FUNCTION_BLOCK FB_StationPLC IMPLEMENTS I_Device, I_Test
VAR_INPUT
END_VAR
VAR_OUTPUT
END_VAR
VAR
END_VAR


// Used to Handhsake Test Controller IPC and Station PLC
mTestStart();
mTestStop();

{warning 'add method implementation '}
METHOD mDeviceComm : BOOL
END_METHOD

{warning 'add method implementation '}
METHOD mDeviceEnable : BOOL
END_METHOD

{warning 'add method implementation '}
METHOD mDeviceHeartbeat : BOOL
END_METHOD

{warning 'add method implementation '}
METHOD mDeviceReset : BOOL
END_METHOD

{warning 'add method implementation '}
METHOD mDeviceStatus : E_DeviceStatus
END_METHOD

{warning 'add method implementation '}
METHOD mTestComp : BOOL
END_METHOD

{warning 'add method implementation '}
METHOD mTestFault : BOOL
END_METHOD

{warning 'add method implementation '}
METHOD mTestResult : BOOL
END_METHOD

{warning 'add method implementation '}
METHOD mTestStart : BOOL
END_METHOD

{warning 'add method implementation '}
METHOD mTestStop : BOOL
END_METHOD

{warning 'add property implementation'}
PROPERTY pDeviceCommOK : BOOL
GET
END_GET
SET
END_SET
END_PROPERTY

{warning 'add property implementation'}
PROPERTY pDeviceEnableCmd : BOOL
GET
END_GET
SET
END_SET
END_PROPERTY

{warning 'add property implementation'}
PROPERTY pDeviceEnabled : BOOL
GET
END_GET
SET
END_SET
END_PROPERTY

{warning 'add property implementation'}
PROPERTY pDeviceFaulted : BOOL
GET
END_GET
SET
END_SET
END_PROPERTY

{warning 'add property implementation'}
PROPERTY pDeviceReady : BOOL
GET
END_GET
SET
END_SET
END_PROPERTY

{warning 'add property implementation'}
PROPERTY pDeviceReset : BOOL
SET
END_SET
END_PROPERTY

{warning 'add property implementation'}
PROPERTY pDeviceStatusFeedback : DWORD
GET
END_GET
SET
END_SET
END_PROPERTY

END_FUNCTION_BLOCK

(* stored: Version 1.1.0.1
   POU FB_StationPLC: Id {c2bbdccd-edf6-4203-96ae-745c9a753c49}, SpecialFunc None
   Method mDeviceComm: Id {6b1c62f9-afd1-0ed1-1af2-c3fcab9e5ac0}
   Method mDeviceEnable: Id {22c773e2-1b2d-0832-05a1-8e46a9989866}
   Method mDeviceHeartbeat: Id {53afa9d6-7a86-02a9-1060-5dfaa73e8c85}
   Method mDeviceReset: Id {19fe8716-a610-0fc6-3d06-68d4d0c31d67}
   Method mDeviceStatus: Id {7e9e7920-bba0-0968-2130-913bdc597fdf}
   Method mTestComp: Id {4402dc0a-65cc-0cc3-0733-13bfaffc6a56}
   Method mTestFault: Id {a285c622-790c-0dc9-2c21-adb29954baa1}
   Method mTestResult: Id {3b83cf7a-caa2-080b-1316-1e6441063419}
   Method mTestStart: Id {d21d38c3-94d0-09be-1e78-d755715e022a}
   Method mTestStop: Id {d3f6af41-3062-0dcd-2377-34ec04c65569}
   Property pDeviceCommOK: Id {4916703a-b0d4-0bb2-3525-62abe97a6292}
   Get Get: Id {e92bb307-03a6-0f96-17bb-7d285d137f4a}
   Set Set: Id {e21a621c-c315-0a6e-3ec6-65b2447003d5}
   Property pDeviceEnableCmd: Id {7e815da2-0217-0362-056d-7bb689a0a5ea}
   Get Get: Id {cb63ff0a-ba88-0941-1472-99edd2723c80}
   Set Set: Id {6d478902-1241-0c40-1479-cd02648cf134}
   Property pDeviceEnabled: Id {6784b490-f0e2-038b-004e-8458e58ffafd}
   Get Get: Id {686c4aef-090b-05dd-3396-43a529d14e88}
   Set Set: Id {08ebb7be-b1cf-08a5-0d5c-80a25b10fbe0}
   Property pDeviceFaulted: Id {25c4060c-f954-008d-06d4-6dea69036e9f}
   Get Get: Id {36ca6899-a424-0799-285c-a2ace000ed00}
   Set Set: Id {5ef681d2-63d6-0ead-2186-e1ab3d7e79b7}
   Property pDeviceReady: Id {2a8f795a-4454-069b-2897-627f8a994a17}
   Get Get: Id {0599777e-dabc-098a-3177-37166d3b8fca}
   Set Set: Id {2fd13787-75ce-0d4d-04c3-e26b54dbab6c}
   Property pDeviceReset: Id {084f9483-9465-0d01-2198-8856abd2a951}
   Set Set: Id {b9c10249-9d7f-0716-11fc-cb7afced8b91}
   Property pDeviceStatusFeedback: Id {94635081-8e06-0d01-2ddb-432446d15997}
   Get Get: Id {26df44a8-ec21-0dee-2432-e3244a0f00e2}
   Set Set: Id {f247035b-e819-06f4-00b3-14bbac8a411d} *)
